# B&R Automation Studio project mappView1
Automation Studio 4.5.2.102; my first mapp view project; technology packages: mappView 5.5.0

## Configuration Config1

CPU PC_any, AutomationRuntime D4.52, Build 4.1.2

### Task classes (Cpu.sw)
```
Cyclic#4:
  Program <- Program.prg
```

### Hardware
```
PC : PC_any v1.1.0.0 (OrderNumber=PC)
  ConfigurationID = mappView1_Config1
  ActivateOpcUa = 1
  OpcUaInformationModels_PV_Version = 1
```

## Logical view

Binary libraries used (declarations not repeated): operator, runtime, astime, AsIecCon

### Package Logical/Libraries - Global libraries

- Visualisation Logical/mappView (not shown)

### Program Logical/Program (IEC)

#### Init.st - Init code
```iecst
PROGRAM _INIT
	Speed := 30;
	Temperature := 20.0;

END_PROGRAM
```

#### Variables.var - Local variables
```iecst
VAR
	Speed : INT;
	Temperature : REAL;
END_VAR
```

Listed in the project but not available here: Logical/Global.typ, Logical/Global.var, Logical/Program/Cyclic.st, Logical/Program/Exit.st, Logical/Program/Types.typ
